// TIA Portal V17 export
// export: Created 2023-12-22T15:03:09.6222836Z, ExportSetting WithDefaults, DisplayName Totally Integrated Automation Portal, DisplayVersion V17, DisplayName TIA Portal Openness, DisplayVersion V17, DisplayName TIA Portal Version Control Interface, DisplayVersion V17, DisplayName STEP 7 Professional, DisplayVersion V17, DisplayName STEP 7 Safety, DisplayVersion V17, DisplayName WinCC Advanced, DisplayVersion V17
DATA_BLOCK "FE_DB"   // DB395
{ S7_Optimized_Access := 'FALSE' }
VERSION : 0.1
// stored: AutoNumber false, DBAccessibleFromOPCUA true, DBAccessibleFromWebserver true, IsOnlyStoredInLoadMemory false, IsWriteProtectedInAS false
   VAR RETAIN
      FE : Array[0..10] of Struct   // Чтение - Input Register (04), Запись - Holding Register (06)
         Flow_Out : Real;   // Накопленный объем +
         Flow_In : Real;   // Накопленный объём -
         Flow : Real;   // Мгновенный расход
         TE_1 : Real;   // Температура канала 1, С
         TE_2 : Real;   // Температура канала 2, С
         PE : Real;   // Давление среды, кПа
         Use { S7_SetPoint := 'True'} : Bool;
         Link : Bool;
         NoRead : Bool;
         NoWrite : Bool;
         ID { S7_SetPoint := 'True'} : Int;
         ADDR { S7_SetPoint := 'True'} : UInt;
         "Name" { S7_SetPoint := 'True'} : String[10];
      END_STRUCT;
   END_VAR
BEGIN
   FE[0].Use := FALSE;
   FE[1..2].Use := TRUE;
   FE[3..10].Use := FALSE;
   FE[0].ID := 0;
   FE[1..2].ID := 14;
   FE[3..10].ID := 0;
   FE[0].ADDR := 0;
   FE[1].ADDR := 41;
   FE[2].ADDR := 42;
   FE[3..10].ADDR := 0;
   FE[0]."Name" := '';
   FE[1]."Name" := 'FE';
   FE[2..10]."Name" := '';
END_DATA_BLOCK
